(* CODESYS project FB_TONR_EXAMPLE_CoDeSys3_3_EXPORT_V2.export

Project tree, tasks and I/O mapping:
  pou TONR [LD]
*)

// TONR

VAR // added by the converter: edge detectors and wires of the graphical bodies
    _w1 : BOOL;
END_VAR

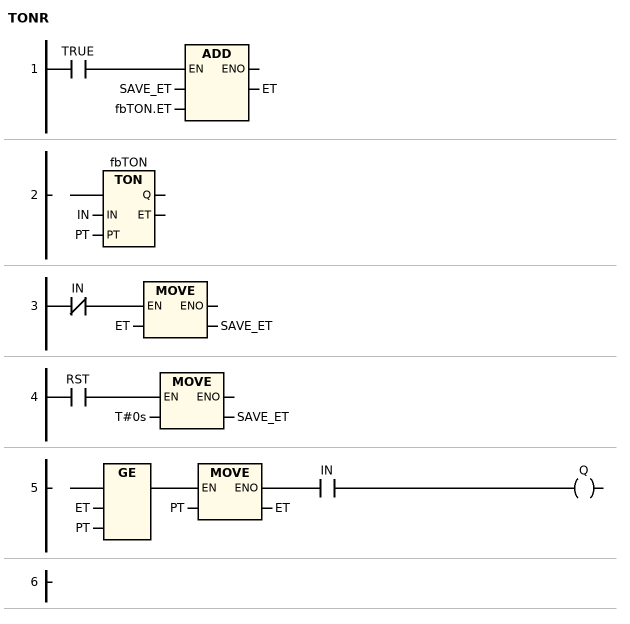
// NETWORK 1
//   fbTON.ET: elapsed time since rising edge at IN
ET := SAVE_ET + fbTON.ET;

// NETWORK 2
fbTON(IN := IN, PT := PT); // TON

// NETWORK 3
IF NOT IN THEN SAVE_ET := ET; END_IF

// NETWORK 4
IF RST THEN SAVE_ET := T#0s; END_IF

// NETWORK 5
_w1 := ET >= PT;
IF _w1 THEN ET := PT; END_IF
Q := _w1 AND IN;

// NETWORK 6
